(* IEC 61131-3 sources: Simple/Grafcet/build (part 2) *)

  STEP Step40:
  END_STEP

  STEP Step44:
    warehouseBusy(R);
    action0(R);
  END_STEP

  TRANSITION FROM Step44 TO Step9
    := true;
  END_TRANSITION

END_PROGRAM

PROGRAM loadProgram
  VAR_EXTERNAL
    isLoadingP1 : BOOL;
    isLoadingP2 : BOOL;
  END_VAR
  VAR
    warehouseIn AT %IW0.0.2.0 : INT;
  END_VAR
  VAR_EXTERNAL
    runFrontCT6_ex : BOOL;
    sensorCT6_ex : BOOL;
    sendRightDownCT2_ex : BOOL;
  END_VAR
  VAR
    sensorAT1 AT %IX0.0.0.0 : BOOL;
    PM AT %IW0.1.1.2 : INT;
  END_VAR
  VAR
    initialPiece : INT;
    finalPiece : INT;
  END_VAR
  VAR_EXTERNAL
    warehouseBusy : BOOL;
    runFrontAT1_ex : BOOL;
    runFrontSaT1_ex : BOOL;
    runFrontSaT2_ex : BOOL;
    runFrontSaT4_ex : BOOL;
    runFrontSbT1_ex : BOOL;
    runFrontSbT2_ex : BOOL;
    runFrontSbT4_ex : BOOL;
    runFrontScT1_ex : BOOL;
    runFrontScT2_ex : BOOL;
    runFrontScT4_ex : BOOL;
    runFrontMT1_ex : BOOL;
    runFrontMT2_ex : BOOL;
    runBackMT5_ex : BOOL;
    runFrontCT1_ex : BOOL;
    runFrontCT3_ex : BOOL;
    runFrontCT4_ex : BOOL;
    runFrontCT5_ex : BOOL;
    runBackSaT7_ex : BOOL;
    runBackScT7_ex : BOOL;
    runBackSbT7_ex : BOOL;
    runBackSbT6_ex : BOOL;
    runBackSaT6_ex : BOOL;
    runBackScT6_ex : BOOL;
    runBackCT9_ex : BOOL;
    runBackCT3_ex : BOOL;
    sendDownSaT2_ex : BOOL;
    sendDownSbT2_ex : BOOL;
    sendDownScT2_ex : BOOL;
    toolPieceSaT3_ex : BOOL;
    toolPieceSaT5_ex : BOOL;
    toolPieceSbT3_ex : BOOL;
    toolPieceSbT5_ex : BOOL;
    toolPieceScT3_ex : BOOL;
    toolPieceScT5_ex : BOOL;
    sendDownCT2_ex : BOOL;
    sensorAT1_ex : BOOL;
    sensorAT2_ex : BOOL;
    sensorSaT1_ex : BOOL;
    sensorSaT2_ex : BOOL;
    sensorSaT3_ex : BOOL;
    sensorSaT4_ex : BOOL;
    sensorSaT5_ex : BOOL;
    sensorSaT6_ex : BOOL;
    sensorSaT7_ex : BOOL;
    sensorSbT1_ex : BOOL;
    sensorSbT2_ex : BOOL;
    sensorSbT3_ex : BOOL;
    sensorSbT4_ex : BOOL;
    sensorSbT5_ex : BOOL;
    sensorSbT6_ex : BOOL;
    sensorSbT7_ex : BOOL;
    sensorScT1_ex : BOOL;
    sensorScT2_ex : BOOL;
    sensorScT3_ex : BOOL;
    sensorScT4_ex : BOOL;
    sensorScT5_ex : BOOL;
    sensorScT6_ex : BOOL;
    sensorScT7_ex : BOOL;
    sensorMT1_ex : BOOL;
    sensorMT2_ex : BOOL;
    sensorCT1_ex : BOOL;
    sensorCT2_ex : BOOL;
    sensorCT3_ex : BOOL;
    sensorCT4_ex : BOOL;
    sensorCT5_ex : BOOL;
    sensorCT7_ex : BOOL;
    sensorCT8_ex : BOOL;
    sensorCT9_ex : BOOL;
    sensorMT6_ex : BOOL;
    sensorMT5_ex : BOOL;
    pushToRollCT4_ex : BOOL;
    pushToRollCT5_ex : BOOL;
    pushToRollCT6_ex : BOOL;
    sendLeftDownSaT6_ex : BOOL;
    sendLeftDownSbT6_ex : BOOL;
    sendLeftDownScT6_ex : BOOL;
    sendLeftDownCT8_ex : BOOL;
    runBackCT8_ex : BOOL;
    runBackMT6_ex : BOOL;
    runBackCT7_ex : BOOL;
    putPieceInSignal_ex : BOOL;
  END_VAR
  VAR
    removeFromWarehouse0 : removeFromWarehouse;
  END_VAR
  VAR
    runUnload AT %IX0.1.0.1 : BOOL;
    runTransformMach1 AT %IX0.1.0.2 : BOOL;
    runTransformMach2 AT %IX0.1.0.3 : BOOL;
    runTransformMach3 AT %IX0.1.0.4 : BOOL;
    cell1Busy AT %QX0.1.0.5 : BOOL;
    cell2Busy AT %QX0.1.0.6 : BOOL;
    cell3Busy AT %QX0.1.0.7 : BOOL;
  END_VAR
  VAR_EXTERNAL
    readyToSendSaT3_ex : BOOL;
    readyToSendSaT5_ex : BOOL;
    readyToSendSbT3_ex : BOOL;
    readyToSendSbT5_ex : BOOL;
    readyToSendScT3_ex : BOOL;
    readyToSendScT5_ex : BOOL;
  END_VAR

  INITIAL_STEP Step7:
  END_STEP

  TRANSITION FROM Step7 TO Step165
    := sensorCT3_ex;
  END_TRANSITION

  STEP Step165:
    runBackCT3_ex(N);
    sendRightDownCT2_ex(N);
    isLoadingP1(S);
  END_STEP

  TRANSITION FROM Step165 TO Step8
    := not sensorCT3_ex;
  END_TRANSITION

  STEP Step8:
  END_STEP

  TRANSITION FROM Step8 TO Step78
    := sensorCT2_ex;
  END_TRANSITION

  STEP Step78:
    runFrontCT4_ex(N);
  END_STEP

  TRANSITION FROM Step78 TO Step79
    := not sensorCT2_ex;
  END_TRANSITION

  STEP Step79:
  END_STEP

  TRANSITION FROM Step79 TO Step80
    := sensorCT4_ex;
  END_TRANSITION

  STEP Step80:
    runFrontCT5_ex(N);
    isLoadingP1(R);
  END_STEP

  TRANSITION FROM Step80 TO Step82
    := not sensorCT4_ex;
  END_TRANSITION

  STEP Step82:
  END_STEP

  TRANSITION FROM Step82 TO Step83
    := sensorCT5_ex;
  END_TRANSITION

  STEP Step83:
    runFrontCT6_ex(N);
  END_STEP

  TRANSITION FROM Step83 TO Step84
    := not sensorCT5_ex;
  END_TRANSITION

  STEP Step84:
  END_STEP

  TRANSITION FROM Step84 TO Step85
    := sensorCT6_ex and (not isLoadingP2);
  END_TRANSITION

  STEP Step85:
    sendLeftDownCT8_ex(N);
  END_STEP

  TRANSITION FROM Step85 TO (Step11, Step12)
    := not sensorCT6_ex;
  END_TRANSITION

  STEP Step11:
  END_STEP

  TRANSITION FROM Step11 TO Step6
    := true;
  END_TRANSITION

  STEP Step6:
  END_STEP

  TRANSITION FROM Step6 TO Step163
    := sensorCT8_ex;
  END_TRANSITION

  STEP Step163:
    runBackCT7_ex(N);
  END_STEP

  TRANSITION FROM Step163 TO Step4
    := not sensorCT8_ex;
  END_TRANSITION

  STEP Step4:
  END_STEP

  TRANSITION FROM Step4 TO Step162
    := sensorCT7_ex;
  END_TRANSITION

  STEP Step162:
    runBackMT6_ex(N);
    isLoadingP2(R);
  END_STEP

  TRANSITION FROM Step162 TO Step3
    := not sensorCT7_ex;
  END_TRANSITION

  STEP Step3:
  END_STEP

  TRANSITION FROM Step3 TO Step161
    := sensorMT6_ex;
  END_TRANSITION

  STEP Step161:
    runBackMT5_ex(N);
  END_STEP

  TRANSITION FROM Step161 TO Step2
    := not sensorMT6_ex;
  END_TRANSITION

  STEP Step2:
  END_STEP

  TRANSITION FROM Step2 TO Step151
    := sensorMT5_ex;
  END_TRANSITION

  STEP Step151:
    runBackScT6_ex(N);
  END_STEP

  TRANSITION FROM Step151 TO Step1
    := not sensorMT5_ex;
  END_TRANSITION

  STEP Step1:
  END_STEP

  TRANSITION FROM Step1 TO Step149
    := sensorScT6_ex;
  END_TRANSITION

  STEP Step149:
    runBackScT7_ex(N);
  END_STEP

  TRANSITION FROM Step149 TO Step0
    := not sensorScT6_ex;
  END_TRANSITION

  STEP Step0:
  END_STEP

  TRANSITION FROM Step0 TO Step147
    := sensorScT7_ex;
  END_TRANSITION

  STEP Step147:
    runBackSbT6_ex(N);
  END_STEP

  TRANSITION FROM Step147 TO Step148
    := not sensorScT7_ex;
  END_TRANSITION

  STEP Step148:
  END_STEP

  TRANSITION FROM Step148 TO Step152
    := sensorSbT6_ex;
  END_TRANSITION

  STEP Step152:
    runBackSbT7_ex(N);
  END_STEP

  TRANSITION FROM Step152 TO Step153
    := not sensorSbT6_ex;
  END_TRANSITION

  STEP Step153:
  END_STEP

  TRANSITION FROM Step153 TO Step154
    := sensorSbT7_ex;
  END_TRANSITION

  STEP Step154:
    runBackSaT6_ex(N);
  END_STEP

  TRANSITION FROM Step154 TO Step156
    := not sensorSbT7_ex;
  END_TRANSITION

  STEP Step156:
  END_STEP

  TRANSITION FROM Step156 TO Step157
    := sensorSaT6_ex;
  END_TRANSITION

  STEP Step157:
    runBackSaT7_ex(N);
  END_STEP

  TRANSITION FROM Step157 TO Step150
    := not sensorSaT6_ex;
  END_TRANSITION

  STEP Step150:
  END_STEP

  TRANSITION FROM Step150 TO Step155
    := sensorSaT7_ex;
  END_TRANSITION

  STEP Step155:
    putPieceInSignal_ex(N);
    cell3Busy(R);
  END_STEP

  TRANSITION FROM Step155 TO Step158
    := not sensorSaT7_ex;
  END_TRANSITION

  STEP Step158:
  END_STEP

  TRANSITION FROM Step158 TO Step159
    := sensorAT2_ex;
  END_TRANSITION

  STEP Step159:
  END_STEP

  TRANSITION FROM Step159 TO Step160
    := not sensorAT2_ex;
  END_TRANSITION

  STEP Step160:
  END_STEP

  STEP Step12:
  END_STEP

  TRANSITION FROM Step12 TO Step7
    := true;
  END_TRANSITION

  INITIAL_STEP Step5:
  END_STEP

  TRANSITION FROM Step5 TO Step164
    := sensorCT9_ex;
  END_TRANSITION

  STEP Step164:
    runBackCT8_ex(N);
    isLoadingP2(S);
    runBackCT9_ex(N);
  END_STEP

  TRANSITION FROM Step164 TO (Step9, Step10)
    := not sensorCT9_ex;
  END_TRANSITION

  STEP Step9:
  END_STEP

  TRANSITION FROM Step9 TO Step6
    := true;
  END_TRANSITION

  STEP Step10:
  END_STEP

  TRANSITION FROM Step10 TO Step5
    := true;
  END_TRANSITION

END_PROGRAM

PROGRAM gantryProgram
  VAR_EXTERNAL
    mounting : BOOL;
    sensorCT7_ex : BOOL;
    pushUpCT6_ex : BOOL;
    runFrontCT7_ex : BOOL;
    sensorCT8_ex : BOOL;
    sendUpRightMT6_ex : BOOL;
    sendRightUpCT8_ex : BOOL;
    runFrontMT3_ex : BOOL;
    runFrontMT4_ex : BOOL;
    sensorCT6_ex : BOOL;
    sensorMT3_ex : BOOL;
    sensorMT4_ex : BOOL;
    sensorMT6_ex : BOOL;
    receivePieceMT1_ex : BOOL;
    receivePieceMT2_ex : BOOL;
    receivePieceMT4_ex : BOOL;
    sendDownMT2_ex : BOOL;
  END_VAR
  VAR
    mount AT %IX0.1.0.8 : BOOL;
  END_VAR
  VAR_EXTERNAL
    gantryBusy_ex : BOOL;
    pickPiece_ex : BOOL;
    releasePiece_ex : BOOL;
    X0Y0_ex : BOOL;
    X0Y1_ex : BOOL;
    X0Y2_ex : BOOL;
    X0Y3_ex : BOOL;
    X0Y4_ex : BOOL;
    X1Y0_ex : BOOL;
    X1Y1_ex : BOOL;
    X1Y2_ex : BOOL;
    X1Y3_ex : BOOL;
    X1Y4_ex : BOOL;
  END_VAR
  VAR
    warehouseIn AT %IW0.0.2.0 : INT;
    sensorAT1 AT %IX0.0.0.0 : BOOL;
    PM AT %IW0.1.1.2 : INT;
    bottomPiece AT %IW0.1.1.5 : INT;
    topPiece AT %IW0.1.1.1 : INT;
  END_VAR
  VAR
    pieceToUnload : INT;
  END_VAR
  VAR
    warehouseBusy AT %QX0.1.0.0 : BOOL;
  END_VAR
  VAR_EXTERNAL
    runFrontAT1_ex : BOOL;
    runFrontSaT1_ex : BOOL;
    runFrontSaT2_ex : BOOL;
    runFrontSaT4_ex : BOOL;
    runFrontSbT1_ex : BOOL;
    runFrontSbT2_ex : BOOL;
    runFrontSbT4_ex : BOOL;
    runFrontScT1_ex : BOOL;
    runFrontScT2_ex : BOOL;
    runFrontScT4_ex : BOOL;
    runFrontMT1_ex : BOOL;
    runFrontMT2_ex : BOOL;
    runFrontCT1_ex : BOOL;
    runFrontCT4_ex : BOOL;
    runFrontCT5_ex : BOOL;
    runBackSaT7_ex : BOOL;
    runBackScT7_ex : BOOL;
    runBackSbT7_ex : BOOL;
    runBackSbT6_ex : BOOL;
    runBackSaT6_ex : BOOL;
    sendDownSaT2_ex : BOOL;
    sendDownSbT2_ex : BOOL;
    sendDownScT2_ex : BOOL;
    toolPieceSaT3_ex : BOOL;
    toolPieceSaT5_ex : BOOL;
    toolPieceSbT3_ex : BOOL;
    toolPieceSbT5_ex : BOOL;
    toolPieceScT3_ex : BOOL;
    toolPieceScT5_ex : BOOL;
    sendDownCT2_ex : BOOL;
    sensorAT1_ex : BOOL;
    sensorAT2_ex : BOOL;
    sensorSaT1_ex : BOOL;
    sensorSaT2_ex : BOOL;
    sensorSaT3_ex : BOOL;
    sensorSaT4_ex : BOOL;
    sensorSaT5_ex : BOOL;
    sensorSaT6_ex : BOOL;
    sensorSaT7_ex : BOOL;
    sensorSbT1_ex : BOOL;
    sensorSbT2_ex : BOOL;
    sensorSbT3_ex : BOOL;
    sensorSbT4_ex : BOOL;
    sensorSbT5_ex : BOOL;
    sensorSbT6_ex : BOOL;
    sensorSbT7_ex : BOOL;
    sensorScT1_ex : BOOL;
    sensorScT2_ex : BOOL;
    sensorScT3_ex : BOOL;
    sensorScT4_ex : BOOL;
    sensorScT5_ex : BOOL;
    sensorScT6_ex : BOOL;
    sensorScT7_ex : BOOL;
    sensorMT1_ex : BOOL;
    sensorMT2_ex : BOOL;
    sensorCT1_ex : BOOL;
    sensorCT2_ex : BOOL;
    sensorCT4_ex : BOOL;
    sensorCT5_ex : BOOL;
    pushToRollCT4_ex : BOOL;
    pushToRollCT5_ex : BOOL;
    pushToRollCT6_ex : BOOL;
    sendLeftDownSaT6_ex : BOOL;
    sendLeftDownSbT6_ex : BOOL;
    sendLeftDownScT6_ex : BOOL;
    putPieceInSignal_ex : BOOL;
  END_VAR
  VAR
    removeFromWarehouse0 : removeFromWarehouse;
  END_VAR
  VAR
    runUnload AT %IX0.1.0.1 : BOOL;
    runTransformMach1 AT %IX0.1.0.2 : BOOL;
    runTransformMach2 AT %IX0.1.0.3 : BOOL;
    runTransformMach3 AT %IX0.1.0.4 : BOOL;
  END_VAR
  VAR_EXTERNAL
    readyToSendSaT3_ex : BOOL;
    readyToSendSaT5_ex : BOOL;
    readyToSendSbT3_ex : BOOL;
    readyToSendSbT5_ex : BOOL;
    readyToSendScT3_ex : BOOL;
    readyToSendScT5_ex : BOOL;
  END_VAR

  INITIAL_STEP Step9:
  END_STEP

  TRANSITION FROM Step9 TO Step30
    := mount and (not warehouseBusy);
  END_TRANSITION

  STEP Step30:
    action0(S);
    warehouseBusy(S);
    unloadBottom(N);
    mount(R);
  END_STEP

  ACTION action0:
    removeFromWarehouse0(pieceNum := pieceToUnload, sensorAT1 := sensorAT1);
    warehouseIn := removeFromWarehouse0.warehouseIn;
  END_ACTION

  ACTION unloadBottom:
    pieceToUnload := bottomPiece;
  END_ACTION

  TRANSITION FROM Step30 TO Step12
    := sensorAT1_ex;
  END_TRANSITION

  STEP Step12:
    runFrontSaT1_ex(N);
    runFrontAT1_ex(N);
  END_STEP

  TRANSITION FROM Step12 TO (Step11, Step14)
    := NOT sensorAT1_ex;
  END_TRANSITION

  STEP Step11:
  END_STEP

  TRANSITION FROM Step11 TO Step10
    := sensorSaT1_ex;
  END_TRANSITION

  STEP Step10:
    runFrontSaT2_ex(N);
  END_STEP

  TRANSITION FROM Step10 TO Step13
    := not sensorSaT1_ex;
  END_TRANSITION

  STEP Step13:
  END_STEP

  TRANSITION FROM Step13 TO Step15
    := sensorSaT2_ex;
  END_TRANSITION

  STEP Step15:
    runFrontSbT1_ex(N);
  END_STEP

  TRANSITION FROM Step15 TO Step16
    := not sensorSaT2_ex;
  END_TRANSITION

  STEP Step16:
  END_STEP

  TRANSITION FROM Step16 TO Step17
    := sensorSbT1_ex;
  END_TRANSITION

  STEP Step17:
    runFrontSbT2_ex(N);
  END_STEP

  TRANSITION FROM Step17 TO Step18
    := not sensorSbT1_ex;
  END_TRANSITION

  STEP Step18:
  END_STEP

  TRANSITION FROM Step18 TO Step19
    := sensorSbT2_ex;
  END_TRANSITION

  STEP Step19:
    runFrontScT1_ex(N);
  END_STEP

  TRANSITION FROM Step19 TO Step20
    := not sensorSbT2_ex;
  END_TRANSITION

  STEP Step20:
  END_STEP

  TRANSITION FROM Step20 TO Step21
    := sensorScT1_ex;
  END_TRANSITION

  STEP Step21:
    runFrontScT2_ex(N);
  END_STEP

  TRANSITION FROM Step21 TO Step22
    := not sensorScT1_ex;
  END_TRANSITION

  STEP Step22:
  END_STEP

  TRANSITION FROM Step22 TO Step23
    := sensorScT2_ex;
  END_TRANSITION

  STEP Step23:
    runFrontMT1_ex(N);
  END_STEP

  TRANSITION FROM Step23 TO Step24
    := not sensorScT2_ex;
  END_TRANSITION

  STEP Step24:
  END_STEP

  TRANSITION FROM Step24 TO Step25
    := sensorMT1_ex;
  END_TRANSITION

  STEP Step25:
    sendDownMT2_ex(N);
  END_STEP

  TRANSITION FROM Step25 TO Step26
    := not sensorMT1_ex;
  END_TRANSITION

  STEP Step26:
  END_STEP

  TRANSITION FROM Step26 TO Step39
    := sensorMT2_ex;
  END_TRANSITION

  STEP Step39:
    runFrontMT3_ex(N);
  END_STEP

  TRANSITION FROM Step39 TO Step53
    := not sensorMT2_ex;
  END_TRANSITION

  STEP Step53:
  END_STEP

  TRANSITION FROM Step53 TO (Step54, Step0)
    := sensorMT3_ex and (not mounting);
  END_TRANSITION

  STEP Step54:
    receivePieceMT4_ex(N);
  END_STEP

  TRANSITION FROM Step54 TO Step56
    := not sensorMT3_ex;
  END_TRANSITION

  STEP Step56:
  END_STEP

  TRANSITION FROM Step56 TO Step55
    := sensorMT4_ex;
  END_TRANSITION

  STEP Step55:
  END_STEP

  TRANSITION FROM (Step55, Step57) TO Step59
    := not gantryBusy_ex;
  END_TRANSITION

  STEP Step59:
    pickPiece_ex(N);
  END_STEP

  TRANSITION FROM Step59 TO Step60
    := gantryBusy_ex;
  END_TRANSITION

  STEP Step60:
  END_STEP

  TRANSITION FROM Step60 TO Step61
    := not gantryBusy_ex;
  END_TRANSITION

  STEP Step61:
    X0Y3_ex(N);
  END_STEP

  TRANSITION FROM Step61 TO Step62
    := gantryBusy_ex;
  END_TRANSITION

  STEP Step62:
  END_STEP

  TRANSITION FROM Step62 TO Step63
    := not gantryBusy_ex;
  END_TRANSITION

  STEP Step63:
    releasePiece_ex(N);
    mounting(S);
  END_STEP

  TRANSITION FROM Step63 TO Step64
    := gantryBusy_ex;
  END_TRANSITION

  STEP Step64:
  END_STEP

  TRANSITION FROM Step64 TO Step88
    := not gantryBusy_ex;
  END_TRANSITION

  STEP Step88:
  END_STEP

  TRANSITION FROM (Step88, Step90) TO Step97
    := not gantryBusy_ex;
  END_TRANSITION

  STEP Step97:
    X1Y3_ex(N);
  END_STEP

  TRANSITION FROM Step97 TO Step98
    := gantryBusy_ex;
  END_TRANSITION

  STEP Step98:
  END_STEP

  TRANSITION FROM Step98 TO Step91
    := not gantryBusy_ex;
  END_TRANSITION

  STEP Step91:
    pickPiece_ex(N);
  END_STEP

  TRANSITION FROM Step91 TO Step92
    := gantryBusy_ex;
  END_TRANSITION

  STEP Step92:
  END_STEP

  TRANSITION FROM Step92 TO Step93
    := not gantryBusy_ex;
  END_TRANSITION

  STEP Step93:
    X0Y3_ex(N);
  END_STEP

  TRANSITION FROM Step93 TO Step94
    := gantryBusy_ex;
  END_TRANSITION

  STEP Step94:
  END_STEP

  TRANSITION FROM Step94 TO Step95
    := not gantryBusy_ex;
  END_TRANSITION

  STEP Step95:
    releasePiece_ex(N);
  END_STEP

  TRANSITION FROM Step95 TO Step96
    := gantryBusy_ex;
  END_TRANSITION

  STEP Step96:
  END_STEP

  TRANSITION FROM Step96 TO Step65
    := not gantryBusy_ex;
  END_TRANSITION

  STEP Step65:
    pickPiece_ex(N);
  END_STEP

  TRANSITION FROM Step65 TO Step66
    := gantryBusy_ex;
  END_TRANSITION

  STEP Step66:
  END_STEP

  TRANSITION FROM Step66 TO Step67
    := not gantryBusy_ex;
  END_TRANSITION

  STEP Step67:
    X1Y3_ex(N);
  END_STEP

  TRANSITION FROM Step67 TO Step68
    := gantryBusy_ex;
  END_TRANSITION

  STEP Step68:
  END_STEP

  TRANSITION FROM Step68 TO Step69
    := not gantryBusy_ex;
  END_TRANSITION

  STEP Step69:
    releasePiece_ex(N);
  END_STEP

  TRANSITION FROM Step69 TO Step70
    := gantryBusy_ex;
  END_TRANSITION

  STEP Step70:
  END_STEP

  TRANSITION FROM Step70 TO Step71
    := not gantryBusy_ex;
  END_TRANSITION

  STEP Step71:
    runFrontMT4_ex(N);
    sendUpRightMT6_ex(N);
  END_STEP

  TRANSITION FROM Step71 TO Step81
    := sensorMT4_ex;
  END_TRANSITION

  STEP Step81:
  END_STEP

  TRANSITION FROM Step81 TO Step82
    := not sensorMT4_ex;
  END_TRANSITION

  STEP Step82:
  END_STEP

  TRANSITION FROM Step82 TO Step72
    := sensorMT6_ex;
  END_TRANSITION

  STEP Step72:
    mounting(R);
  END_STEP

  TRANSITION FROM Step72 TO Step73
    := not sensorMT6_ex;
  END_TRANSITION

  STEP Step73:
    runFrontCT7_ex(N);
  END_STEP

  TRANSITION FROM Step73 TO Step74
    := sensorCT7_ex;
  END_TRANSITION

  STEP Step74:
    sendRightUpCT8_ex(N);
  END_STEP

  TRANSITION FROM Step74 TO Step75
    := not sensorCT7_ex;
  END_TRANSITION

  STEP Step75:
  END_STEP

  TRANSITION FROM Step75 TO Step76
    := sensorCT8_ex;
  END_TRANSITION

  STEP Step76:
  END_STEP

  TRANSITION FROM Step76 TO Step77
    := not sensorCT8_ex;
  END_TRANSITION

  STEP Step77:
    pushUpCT6_ex(N);
  END_STEP

  TRANSITION FROM Step77 TO Step79
    := sensorCT6_ex;
  END_TRANSITION

  STEP Step79:
  END_STEP

  TRANSITION FROM Step79 TO Step80
    := not sensorCT6_ex;
  END_TRANSITION

  STEP Step80:
  END_STEP

  TRANSITION FROM Step80 TO Step78
    := true;
  END_TRANSITION

  STEP Step78:
  END_STEP

  STEP Step0:
  END_STEP

  TRANSITION FROM Step0 TO Step58
    := not gantryBusy_ex;
  END_TRANSITION

  STEP Step58:
    X1Y3_ex(N);
  END_STEP

  TRANSITION FROM Step58 TO Step1
    := gantryBusy_ex;
  END_TRANSITION

  STEP Step1:
  END_STEP

  TRANSITION FROM Step1 TO Step57
    := not gantryBusy_ex;
  END_TRANSITION

  STEP Step57:
  END_STEP

  STEP Step14:
    unloadTop(N);
    action0(R);
  END_STEP

  ACTION unloadTop:
    pieceToUnload := topPiece;
  END_ACTION

  TRANSITION FROM Step14 TO sendTop
    := true;
  END_TRANSITION

  STEP sendTop:
    action0(S);
  END_STEP

  TRANSITION FROM sendTop TO Step28
    := sensorAT1_ex;
  END_TRANSITION

  STEP Step28:
    runFrontSaT1_ex(N);
    runFrontAT1_ex(N);
  END_STEP

  TRANSITION FROM Step28 TO (Step42, Step44)
    := NOT sensorAT1_ex;
  END_TRANSITION

  STEP Step42:
  END_STEP

  TRANSITION FROM Step42 TO Step41
    := sensorSaT1_ex;
  END_TRANSITION

  STEP Step41:
    runFrontSaT2_ex(N);
  END_STEP

  TRANSITION FROM Step41 TO Step43
    := not sensorSaT1_ex;
  END_TRANSITION

  STEP Step43:
  END_STEP

  TRANSITION FROM Step43 TO Step45
    := sensorSaT2_ex;
  END_TRANSITION

  STEP Step45:
    runFrontSbT1_ex(N);
  END_STEP

  TRANSITION FROM Step45 TO Step29
    := not sensorSaT2_ex;
  END_TRANSITION

  STEP Step29:
  END_STEP

  TRANSITION FROM Step29 TO Step31
    := sensorSbT1_ex;
  END_TRANSITION

  STEP Step31:
    runFrontSbT2_ex(N);
  END_STEP

  TRANSITION FROM Step31 TO Step32
    := not sensorSbT1_ex;
  END_TRANSITION

  STEP Step32:
  END_STEP

  TRANSITION FROM Step32 TO Step33
    := sensorSbT2_ex;
  END_TRANSITION

  STEP Step33:
    runFrontScT1_ex(N);
  END_STEP

  TRANSITION FROM Step33 TO Step34
    := not sensorSbT2_ex;
  END_TRANSITION

  STEP Step34:
  END_STEP

  TRANSITION FROM Step34 TO Step35
    := sensorScT1_ex;
  END_TRANSITION

  STEP Step35:
    runFrontScT2_ex(N);
  END_STEP

  TRANSITION FROM Step35 TO Step36
    := not sensorScT1_ex;
  END_TRANSITION

  STEP Step36:
  END_STEP

  TRANSITION FROM Step36 TO Step37
    := sensorScT2_ex;
  END_TRANSITION

  STEP Step37:
    runFrontMT1_ex(N);
  END_STEP

  TRANSITION FROM Step37 TO Step38
    := not sensorScT2_ex;
  END_TRANSITION

  STEP Step38:
  END_STEP

  TRANSITION FROM Step38 TO Step40
    := sensorMT1_ex;
  END_TRANSITION

  STEP Step40:
    sendDownMT2_ex(N);
  END_STEP

  TRANSITION FROM Step40 TO Step84
    := not sensorMT1_ex;
  END_TRANSITION

  STEP Step84:
  END_STEP

  TRANSITION FROM Step84 TO Step85
    := sensorMT2_ex;
  END_TRANSITION

  STEP Step85:
    runFrontMT3_ex(N);
  END_STEP

  TRANSITION FROM Step85 TO Step86
    := not sensorMT2_ex;
  END_TRANSITION

  STEP Step86:
  END_STEP

  TRANSITION FROM Step86 TO Step87
    := sensorMT3_ex and (not mounting);
  END_TRANSITION

  STEP Step87:
    receivePieceMT4_ex(N);
  END_STEP

  TRANSITION FROM Step87 TO Step89
    := not sensorMT3_ex;
  END_TRANSITION

  STEP Step89:
  END_STEP

  TRANSITION FROM Step89 TO Step90
    := sensorMT4_ex;
  END_TRANSITION

  STEP Step90:
  END_STEP

  STEP Step44:
    warehouseBusy(R);
  END_STEP

  TRANSITION FROM Step44 TO Step83
    := true;
  END_TRANSITION

  STEP Step83:
    action0(R);
  END_STEP

  TRANSITION FROM Step83 TO Step9
    := true;
  END_TRANSITION

END_PROGRAM

PROGRAM unloadProgram
  VAR_EXTERNAL
    isLoadingP1 : BOOL;
    pieceNum : INT;
    takePiece : BOOL;
  END_VAR
  VAR
    warehouseIn AT %IW0.0.2.0 : INT;
    sensorAT1 AT %IX0.0.0.0 : BOOL;
    PM AT %IW0.1.1.2 : INT;
    initialPiece AT %IW0.1.1.0 : INT;
    finalPiece AT %IW0.1.1.3 : INT;
    warehouseBusy AT %IX0.1.0.0 : BOOL;
  END_VAR
  VAR_EXTERNAL
    runFrontAT1_ex : BOOL;
    runFrontSaT1_ex : BOOL;
    runFrontSaT2_ex : BOOL;
    runFrontSaT4_ex : BOOL;
    runFrontSbT1_ex : BOOL;
    runFrontSbT2_ex : BOOL;
    runFrontSbT4_ex : BOOL;
    runFrontScT1_ex : BOOL;
    runFrontScT2_ex : BOOL;
    runFrontScT4_ex : BOOL;
    runFrontMT1_ex : BOOL;
    runFrontMT2_ex : BOOL;
    runFrontCT1_ex : BOOL;
    runFrontCT4_ex : BOOL;
    runFrontCT5_ex : BOOL;
    runBackSaT7_ex : BOOL;
    runBackScT7_ex : BOOL;
    runBackSbT7_ex : BOOL;
    runBackSbT6_ex : BOOL;
    runBackSaT6_ex : BOOL;
    sendDownSaT2_ex : BOOL;
    sendDownSbT2_ex : BOOL;
    sendDownScT2_ex : BOOL;
    toolPieceSaT3_ex : BOOL;
    toolPieceSaT5_ex : BOOL;
    toolPieceSbT3_ex : BOOL;
    toolPieceSbT5_ex : BOOL;
    toolPieceScT3_ex : BOOL;
    toolPieceScT5_ex : BOOL;
    sendDownCT2_ex : BOOL;
    sensorAT1_ex : BOOL;
    sensorAT2_ex : BOOL;
    sensorSaT1_ex : BOOL;
    sensorSaT2_ex : BOOL;
    sensorSaT3_ex : BOOL;
    sensorSaT4_ex : BOOL;
    sensorSaT5_ex : BOOL;
    sensorSaT6_ex : BOOL;
    sensorSaT7_ex : BOOL;
    sensorSbT1_ex : BOOL;
    sensorSbT2_ex : BOOL;
    sensorSbT3_ex : BOOL;
    sensorSbT4_ex : BOOL;
    sensorSbT5_ex : BOOL;
    sensorSbT6_ex : BOOL;
    sensorSbT7_ex : BOOL;
    sensorScT1_ex : BOOL;
    sensorScT2_ex : BOOL;
    sensorScT3_ex : BOOL;
    sensorScT4_ex : BOOL;
    sensorScT5_ex : BOOL;
    sensorScT6_ex : BOOL;
    sensorScT7_ex : BOOL;
    sensorMT1_ex : BOOL;
    sensorMT2_ex : BOOL;
    sensorCT1_ex : BOOL;
    sensorCT2_ex : BOOL;
    sensorCT3_ex : BOOL;
    sensorCT4_ex : BOOL;
    sensorCT5_ex : BOOL;
    sensorCT6_ex : BOOL;
    pushToRollCT4_ex : BOOL;
    pushToRollCT5_ex : BOOL;
    pushToRollCT6_ex : BOOL;
    sendLeftDownSaT6_ex : BOOL;
    sendLeftDownSbT6_ex : BOOL;
    sendLeftDownScT6_ex : BOOL;
    putPieceInSignal_ex : BOOL;
  END_VAR
  VAR
    removeFromWarehouse0 : removeFromWarehouse;
  END_VAR
  VAR
    runUnload AT %IX0.1.0.1 : BOOL;
    runTransformMach1 AT %IX0.1.0.2 : BOOL;
    runTransformMach2 AT %IX0.1.0.3 : BOOL;
    runTransformMach3 AT %IX0.1.0.4 : BOOL;
  END_VAR
  VAR_EXTERNAL
    readyToSendSaT3_ex : BOOL;
    readyToSendSaT5_ex : BOOL;
    readyToSendSbT3_ex : BOOL;
    readyToSendSbT5_ex : BOOL;
    readyToSendScT3_ex : BOOL;
    readyToSendScT5_ex : BOOL;
  END_VAR

  INITIAL_STEP Step0:
  END_STEP

  TRANSITION FROM Step0 TO Step52
    := runUnload AND (not warehouseBusy);
  END_TRANSITION

  STEP Step52:
    warehouseBusy(S);
    runUnload(R);
  END_STEP

  TRANSITION FROM Step52 TO Step26
    := PM = 1;
  END_TRANSITION

  STEP Step26:
    action0(S);
  END_STEP

  ACTION action0:
    removeFromWarehouse0(pieceNum := initialPiece, sensorAT1 := sensorAT1);
    warehouseIn := removeFromWarehouse0.warehouseIn;
  END_ACTION

  TRANSITION FROM Step26 TO Step2
    := sensorAT1_ex;
  END_TRANSITION

  STEP Step2:
    runFrontSaT1_ex(N);
    runFrontAT1_ex(N);
  END_STEP

  TRANSITION FROM Step2 TO Step4
    := NOT sensorAT1_ex;
  END_TRANSITION

  STEP Step4:
    action0(R);
  END_STEP

  TRANSITION FROM Step4 TO (Step3, Step6)
    := sensorSaT1_ex;
  END_TRANSITION

  STEP Step3:
    runFrontSaT2_ex(N);
  END_STEP

  TRANSITION FROM Step3 TO Step5
    := not sensorSaT1_ex;
  END_TRANSITION

  STEP Step5:
  END_STEP

  TRANSITION FROM Step5 TO Step7
    := sensorSaT2_ex;
  END_TRANSITION

  STEP Step7:
    runFrontSbT1_ex(N);
  END_STEP

  TRANSITION FROM Step7 TO Step8
    := not sensorSaT2_ex;
  END_TRANSITION

  STEP Step8:
  END_STEP

  TRANSITION FROM Step8 TO Step9
    := sensorSbT1_ex;
  END_TRANSITION

  STEP Step9:
    runFrontSbT2_ex(N);
  END_STEP

  TRANSITION FROM Step9 TO Step10
    := not sensorSbT1_ex;
  END_TRANSITION

  STEP Step10:
  END_STEP

  TRANSITION FROM Step10 TO Step11
    := sensorSbT2_ex;
  END_TRANSITION

  STEP Step11:
    runFrontScT1_ex(N);
  END_STEP

  TRANSITION FROM Step11 TO Step12
    := not sensorSbT2_ex;
  END_TRANSITION

  STEP Step12:
  END_STEP

  TRANSITION FROM Step12 TO Step13
    := sensorScT1_ex;
  END_TRANSITION

  STEP Step13:
    runFrontScT2_ex(N);
  END_STEP

  TRANSITION FROM Step13 TO Step14
    := not sensorScT1_ex;
  END_TRANSITION

  STEP Step14:
  END_STEP

  TRANSITION FROM Step14 TO Step15
    := sensorScT2_ex;
  END_TRANSITION

  STEP Step15:
    runFrontMT1_ex(N);
  END_STEP

  TRANSITION FROM Step15 TO Step16
    := not sensorScT2_ex;
  END_TRANSITION

  STEP Step16:
  END_STEP

  TRANSITION FROM Step16 TO Step17
    := sensorMT1_ex;
  END_TRANSITION

  STEP Step17:
    runFrontMT2_ex(N);
  END_STEP

  TRANSITION FROM Step17 TO Step18
    := not sensorMT1_ex;
  END_TRANSITION

  STEP Step18:
  END_STEP

  TRANSITION FROM Step18 TO Step19
    := sensorMT2_ex;
  END_TRANSITION

  STEP Step19:
    runFrontCT1_ex(N);
  END_STEP

  TRANSITION FROM Step19 TO Step20
    := not sensorMT2_ex;
  END_TRANSITION

  STEP Step20:
  END_STEP

  TRANSITION FROM Step20 TO Step21
    := sensorCT1_ex AND (not isLoadingP1) AND (not sensorCT3_ex);
  END_TRANSITION

  STEP Step21:
    sendDownCT2_ex(N);
  END_STEP

  TRANSITION FROM Step21 TO Step22
    := not sensorCT1_ex;
  END_TRANSITION

  STEP Step22:
  END_STEP

  TRANSITION FROM Step22 TO Step23
    := sensorCT2_ex;
  END_TRANSITION

  STEP Step23:
    pushToRollCT4_ex(N);
  END_STEP

  TRANSITION FROM Step23 TO Step24
    := not sensorCT2_ex;
  END_TRANSITION

  STEP Step24:
  END_STEP

  TRANSITION FROM Step24 TO Step25
    := sensorCT4_ex;
  END_TRANSITION

  STEP Step25:
  END_STEP

  TRANSITION FROM Step25 TO Step1
    := not sensorCT4_ex;
  END_TRANSITION

  STEP Step1:
  END_STEP

  TRANSITION FROM Step1 TO Step85
    := true;
  END_TRANSITION

  STEP Step85:
  END_STEP

  STEP Step6:
    warehouseBusy(R);
  END_STEP

  TRANSITION FROM Step6 TO Step0
    := true;
  END_TRANSITION

  TRANSITION FROM Step52 TO Step47
    := PM = 2;
  END_TRANSITION

  STEP Step47:
    action0(S);
  END_STEP

  TRANSITION FROM Step47 TO Step46
    := sensorAT1_ex;
  END_TRANSITION

  STEP Step46:
    runFrontSaT1_ex(N);
    runFrontAT1_ex(N);
  END_STEP

  TRANSITION FROM Step46 TO Step28
    := NOT sensorAT1_ex;
  END_TRANSITION

  STEP Step28:
    action0(R);
  END_STEP

  TRANSITION FROM Step28 TO (Step27, Step30)
    := sensorSaT1_ex;
  END_TRANSITION

  STEP Step27:
    runFrontSaT2_ex(N);
  END_STEP

  TRANSITION FROM Step27 TO Step29
    := not sensorSaT1_ex;
  END_TRANSITION

  STEP Step29:
  END_STEP

  TRANSITION FROM Step29 TO Step31
    := sensorSaT2_ex;
  END_TRANSITION

  STEP Step31:
    runFrontSbT1_ex(N);
  END_STEP

  TRANSITION FROM Step31 TO Step32
    := not sensorSaT2_ex;
  END_TRANSITION

  STEP Step32:
  END_STEP

  TRANSITION FROM Step32 TO Step33
    := sensorSbT1_ex;
  END_TRANSITION

  STEP Step33:
    runFrontSbT2_ex(N);
  END_STEP

  TRANSITION FROM Step33 TO Step34
    := not sensorSbT1_ex;
  END_TRANSITION

  STEP Step34:
  END_STEP

  TRANSITION FROM Step34 TO Step35
    := sensorSbT2_ex;
  END_TRANSITION

  STEP Step35:
    runFrontScT1_ex(N);
  END_STEP

  TRANSITION FROM Step35 TO Step36
    := not sensorSbT2_ex;
  END_TRANSITION

  STEP Step36:
  END_STEP

  TRANSITION FROM Step36 TO Step37
    := sensorScT1_ex;
  END_TRANSITION

  STEP Step37:
    runFrontScT2_ex(N);
  END_STEP

  TRANSITION FROM Step37 TO Step38
    := not sensorScT1_ex;
  END_TRANSITION

  STEP Step38:
  END_STEP

  TRANSITION FROM Step38 TO Step39
    := sensorScT2_ex;
  END_TRANSITION

  STEP Step39:
    runFrontMT1_ex(N);
  END_STEP

  TRANSITION FROM Step39 TO Step40
    := not sensorScT2_ex;
  END_TRANSITION

  STEP Step40:
  END_STEP

  TRANSITION FROM Step40 TO Step41
    := sensorMT1_ex;
  END_TRANSITION

  STEP Step41:
    runFrontMT2_ex(N);
  END_STEP

  TRANSITION FROM Step41 TO Step42
    := not sensorMT1_ex;
  END_TRANSITION

  STEP Step42:
  END_STEP

  TRANSITION FROM Step42 TO Step43
    := sensorMT2_ex;
  END_TRANSITION

  STEP Step43:
    runFrontCT1_ex(N);
  END_STEP

  TRANSITION FROM Step43 TO Step44
    := not sensorMT2_ex;
  END_TRANSITION

  STEP Step44:
  END_STEP

  TRANSITION FROM Step44 TO Step45
    := sensorCT1_ex AND (not isLoadingP1) AND (not sensorCT3_ex);
  END_TRANSITION

  STEP Step45:
    sendDownCT2_ex(N);
  END_STEP

  TRANSITION FROM Step45 TO Step48
    := not sensorCT1_ex;
  END_TRANSITION

  STEP Step48:
  END_STEP

  TRANSITION FROM Step48 TO Step49
    := sensorCT2_ex;
  END_TRANSITION

  STEP Step49:
    runFrontCT4_ex(N);
  END_STEP

  TRANSITION FROM Step49 TO Step50
    := not sensorCT2_ex;
  END_TRANSITION

  STEP Step50:
  END_STEP

  TRANSITION FROM Step50 TO Step51
    := sensorCT4_ex;
  END_TRANSITION

  STEP Step51:
    pushToRollCT5_ex(N);
  END_STEP

  TRANSITION FROM Step51 TO Step53
    := not sensorCT4_ex;
  END_TRANSITION

  STEP Step53:
  END_STEP

  TRANSITION FROM Step53 TO Step54
    := sensorCT5_ex;
  END_TRANSITION

  STEP Step54:
  END_STEP

  TRANSITION FROM Step54 TO Step55
    := not sensorCT5_ex;
  END_TRANSITION

  STEP Step55:
  END_STEP

  TRANSITION FROM Step55 TO Step85
    := true;
  END_TRANSITION

  STEP Step30:
    warehouseBusy(R);
  END_STEP

  TRANSITION FROM Step30 TO Step0
    := true;
  END_TRANSITION

  TRANSITION FROM Step52 TO Step80
    := PM = 3;
  END_TRANSITION

  STEP Step80:
    action0(S);
  END_STEP

  TRANSITION FROM Step80 TO Step58
    := sensorAT1_ex;
  END_TRANSITION

  STEP Step58:
    runFrontSaT1_ex(N);
    runFrontAT1_ex(N);
  END_STEP

  TRANSITION FROM Step58 TO Step57
    := NOT sensorAT1_ex;
  END_TRANSITION

  STEP Step57:
    action0(R);
  END_STEP

  TRANSITION FROM Step57 TO (Step56, Step60)
    := sensorSaT1_ex;
  END_TRANSITION

  STEP Step56:
    runFrontSaT2_ex(N);
  END_STEP

  TRANSITION FROM Step56 TO Step59
    := not sensorSaT1_ex;
  END_TRANSITION

  STEP Step59:
  END_STEP

  TRANSITION FROM Step59 TO Step61
    := sensorSaT2_ex;
  END_TRANSITION

  STEP Step61:
    runFrontSbT1_ex(N);
  END_STEP

  TRANSITION FROM Step61 TO Step62
    := not sensorSaT2_ex;
  END_TRANSITION

  STEP Step62:
  END_STEP

  TRANSITION FROM Step62 TO Step63
    := sensorSbT1_ex;
  END_TRANSITION

  STEP Step63:
    runFrontSbT2_ex(N);
  END_STEP

  TRANSITION FROM Step63 TO Step64
    := not sensorSbT1_ex;
  END_TRANSITION

  STEP Step64:
  END_STEP

  TRANSITION FROM Step64 TO Step65
    := sensorSbT2_ex;
  END_TRANSITION

  STEP Step65:
    runFrontScT1_ex(N);
  END_STEP

  TRANSITION FROM Step65 TO Step66
    := not sensorSbT2_ex;
  END_TRANSITION

  STEP Step66:
  END_STEP

  TRANSITION FROM Step66 TO Step67
    := sensorScT1_ex;
  END_TRANSITION

  STEP Step67:
    runFrontScT2_ex(N);
  END_STEP

  TRANSITION FROM Step67 TO Step68
    := not sensorScT1_ex;
  END_TRANSITION

  STEP Step68:
  END_STEP

  TRANSITION FROM Step68 TO Step69
    := sensorScT2_ex;
  END_TRANSITION

  STEP Step69:
    runFrontMT1_ex(N);
  END_STEP

  TRANSITION FROM Step69 TO Step70
    := not sensorScT2_ex;
  END_TRANSITION

  STEP Step70:
  END_STEP

  TRANSITION FROM Step70 TO Step71
    := sensorMT1_ex;
  END_TRANSITION

  STEP Step71:
    runFrontMT2_ex(N);
  END_STEP

  TRANSITION FROM Step71 TO Step72
    := not sensorMT1_ex;
  END_TRANSITION

  STEP Step72:
  END_STEP

  TRANSITION FROM Step72 TO Step73
    := sensorMT2_ex;
  END_TRANSITION

  STEP Step73:
    runFrontCT1_ex(N);
  END_STEP

  TRANSITION FROM Step73 TO Step74
    := not sensorMT2_ex;
  END_TRANSITION

  STEP Step74:
  END_STEP

  TRANSITION FROM Step74 TO Step75
    := sensorCT1_ex AND (not isLoadingP1) AND (not sensorCT3_ex);
  END_TRANSITION

  STEP Step75:
    sendDownCT2_ex(N);
  END_STEP

  TRANSITION FROM Step75 TO Step76
    := not sensorCT1_ex;
  END_TRANSITION

  STEP Step76:
  END_STEP

  TRANSITION FROM Step76 TO Step77
    := sensorCT2_ex;
  END_TRANSITION

  STEP Step77:
    runFrontCT4_ex(N);
  END_STEP

  TRANSITION FROM Step77 TO Step78
    := not sensorCT2_ex;
  END_TRANSITION

  STEP Step78:
  END_STEP

  TRANSITION FROM Step78 TO Step79
    := sensorCT4_ex;
  END_TRANSITION

  STEP Step79:
    runFrontCT5_ex(N);
  END_STEP

  TRANSITION FROM Step79 TO Step81
    := not sensorCT4_ex;
  END_TRANSITION

  STEP Step81:
  END_STEP

  TRANSITION FROM Step81 TO Step82
    := sensorCT5_ex;
  END_TRANSITION

  STEP Step82:
    pushToRollCT6_ex(N);
  END_STEP

  TRANSITION FROM Step82 TO Step83
    := not sensorCT5_ex;
  END_TRANSITION

  STEP Step83:
  END_STEP

  TRANSITION FROM Step83 TO Step84
    := sensorCT6_ex;
  END_TRANSITION

  STEP Step84:
  END_STEP

  TRANSITION FROM Step84 TO Step85
    := not sensorCT6_ex;
  END_TRANSITION

  STEP Step60:
    warehouseBusy(R);
  END_STEP

  TRANSITION FROM Step60 TO Step0
    := true;
  END_TRANSITION

END_PROGRAM

CONFIGURATION config
  VAR_GLOBAL
    mounting : BOOL;
    isLoadingP1 : BOOL;
    isLoadingP2 : BOOL;
    pushUpCT6_ex : BOOL;
    sendRightDownCT2_ex : BOOL;
    sendRightUpCT8_ex : BOOL;
    runFrontCT7_ex : BOOL;
    receivePieceMT3_ex : BOOL;
    sendUpRightMT6_ex : BOOL;
    receivePieceMT4_ex : BOOL;
    sensorMT3_ex : BOOL;
    sensorMT4_ex : BOOL;
    runFrontMT3_ex : BOOL;
    runFrontMT4_ex : BOOL;
    takePiece : BOOL;
    pieceNum : INT;
    cell1Initial : INT;
    cell1Final : INT;
    cell2Initial : INT;
    cell2Final : INT;
    cell3Initial : INT;
    cell3Final : INT;
    receivePieceMT1_ex : BOOL;
    receivePieceMT2_ex : BOOL;
    waitForOp_ex : BOOL;
    ii : BOOL;
    pickPiece_ex : BOOL;
    releasePiece_ex : BOOL;
    X0Y0_ex : BOOL;
    X0Y1_ex : BOOL;
    X0Y2_ex : BOOL;
    X0Y3_ex : BOOL;
    X0Y4_ex : BOOL;
    X1Y0_ex : BOOL;
    X1Y1_ex : BOOL;
    X1Y2_ex : BOOL;
    X1Y3_ex : BOOL;
    X1Y4_ex : BOOL;
    warehouseBusy : BOOL;
    pushToRollCT4_ex : BOOL;
    pushToRollCT5_ex : BOOL;
    pushToRollCT6_ex : BOOL;
    runFrontAT1_ex : BOOL;
    runFrontSaT1_ex : BOOL;
    runFrontSaT2_ex : BOOL;
    runFrontSbT1_ex : BOOL;
    runFrontSbT2_ex : BOOL;
    runFrontScT1_ex : BOOL;
    runFrontScT2_ex : BOOL;
    runFrontMT1_ex : BOOL;
    runFrontMT2_ex : BOOL;
    runFrontCT1_ex : BOOL;
    runFrontCT2_ex : BOOL;
    runFrontCT3_ex : BOOL;
    runBackCT2_ex : BOOL;
    runBackCT3_ex : BOOL;
    sendDownSaT2_ex : BOOL;
    sendDownSbT2_ex : BOOL;
    sendDownScT2_ex : BOOL;
    sendDownMT2_ex : BOOL;
    sendDownCT2_ex : BOOL;
    sendLeftDownSaT6_ex : BOOL;
    sendLeftDownSbT6_ex : BOOL;
    sendLeftDownScT6_ex : BOOL;
    sendLeftDownCT8_ex : BOOL;
    sensorAT1_ex : BOOL;
    sensorSaT1_ex : BOOL;
    sensorSaT2_ex : BOOL;
    sensorSaT3_ex : BOOL;
    sensorSaT4_ex : BOOL;
    sensorSaT5_ex : BOOL;
    sensorSaT6_ex : BOOL;
    sensorSaT7_ex : BOOL;
    sensorSbT1_ex : BOOL;
    sensorSbT2_ex : BOOL;
    sensorSbT3_ex : BOOL;
    sensorSbT4_ex : BOOL;
    sensorSbT5_ex : BOOL;
    sensorSbT6_ex : BOOL;
    sensorSbT7_ex : BOOL;
    sensorScT1_ex : BOOL;
    sensorScT2_ex : BOOL;
    sensorScT3_ex : BOOL;
    sensorScT4_ex : BOOL;
    sensorScT5_ex : BOOL;
    sensorScT6_ex : BOOL;
    sensorScT7_ex : BOOL;
    sensorMT1_ex : BOOL;
    sensorMT2_ex : BOOL;
    sensorCT1_ex : BOOL;
    sensorCT2_ex : BOOL;
    sensorCT3_ex : BOOL;
    sensorCT4_ex : BOOL;
    sensorCT5_ex : BOOL;
    sensorCT6_ex : BOOL;
    sensorAT2_ex : BOOL;
    sensorMT5_ex : BOOL;
    sensorMT6_ex : BOOL;
    sensorCT7_ex : BOOL;
    sensorCT8_ex : BOOL;
    sensorCT9_ex : BOOL;
    sendDownSaT6_ex : BOOL;
    sendDownSbT6_ex : BOOL;
    sendDownScT6_ex : BOOL;
    sendDownMT6_ex : BOOL;
    sendDownCT8_ex : BOOL;
    runBackAT2_ex : BOOL;
    runBackSaT6_ex : BOOL;
    runBackSaT7_ex : BOOL;
    runBackSbT6_ex : BOOL;
    runBackSbT7_ex : BOOL;
    runBackScT6_ex : BOOL;
    runBackScT7_ex : BOOL;
    sendUpSaT6_ex : BOOL;
    runFrontSbT3_ex : BOOL;
    runFrontSbT4_ex : BOOL;
    runFrontSbT5_ex : BOOL;
    runFrontSbT6_ex : BOOL;
    runFrontSaT3_ex : BOOL;
    runFrontSaT4_ex : BOOL;
    runFrontSaT5_ex : BOOL;
    runFrontScT3_ex : BOOL;
    runFrontScT4_ex : BOOL;
    runFrontScT5_ex : BOOL;
    runFrontScT6_ex : BOOL;
    runBackMT5_ex : BOOL;
    runBackMT6_ex : BOOL;
    runBackCT7_ex : BOOL;
    runBackCT8_ex : BOOL;
    runFrontCT8_ex : BOOL;
    runFrontCT4_ex : BOOL;
    runFrontCT5_ex : BOOL;
    runFrontCT6_ex : BOOL;
    runBackCT9_ex : BOOL;
    toolPieceSaT3_ex : BOOL;
    toolPieceSaT5_ex : BOOL;
    toolPieceSbT3_ex : BOOL;
    toolPieceSbT5_ex : BOOL;
    toolPieceScT3_ex : BOOL;
    toolPieceScT5_ex : BOOL;
    readyToSendSaT3_ex : BOOL;
    readyToSendSaT5_ex : BOOL;
    readyToSendSbT5_ex : BOOL;
    readyToSendSbT3_ex : BOOL;
    readyToSendScT3_ex : BOOL;
    readyToSendScT5_ex : BOOL;
    putPieceInSignal_ex : BOOL;
    gantryBusy_ex : BOOL;
  END_VAR

  RESOURCE resource1 ON PLC
    TASK task0(INTERVAL := T#20ms,PRIORITY := 0);
    PROGRAM instance0 WITH task0 : factoryFloorProgram;
    PROGRAM instance3 WITH task0 : gantryProgram;
    PROGRAM instance1 WITH task0 : unloadProgram;
    PROGRAM instance2 WITH task0 : transformProgram;
    PROGRAM instance4 WITH task0 : loadProgram;
  END_RESOURCE
END_CONFIGURATION
